// TIA Portal V17 export
// export: Created 2024-06-14T09:52:32.4574024Z, ExportSetting WithDefaults, DisplayName Totally Integrated Automation Portal, DisplayVersion V17, DisplayName TIA Portal Openness, DisplayVersion V17, DisplayName TIA Portal Version Control Interface, DisplayVersion V17, DisplayName Simotion SCOUT TIA, DisplayVersion 5.4.3.0, DisplayName SINAMICS Startdrive Advanced, DisplayVersion V17 SP1 Update 1, DisplayName SINAMICS Startdrive G110M, G120, G120C, G120D, G120P, G115D, DisplayVersion V17 SP1 Update 1, DisplayName SINAMICS Startdrive G130, G150, S120, S150, SINAMICS MV, S210, DisplayVersion V17 SP1 Update 1, DisplayName STEP 7 Professional, DisplayVersion V17, DisplayName STEP 7 Safety, DisplayVersion V17, DisplayName WinCC Professional, DisplayVersion V17
FUNCTION "MODTCP_STN5_FC_L2" : Void   // FC101, LAD
{ S7_Optimized_Access := 'TRUE' }
VERSION : 0.1
// stored: AutoNumber false, IsIECCheckEnabled false, SetENOAutomatically false, UDAEnableTagReadback false
BEGIN

REGION Network 2: Call Filling Line-1 Station-1
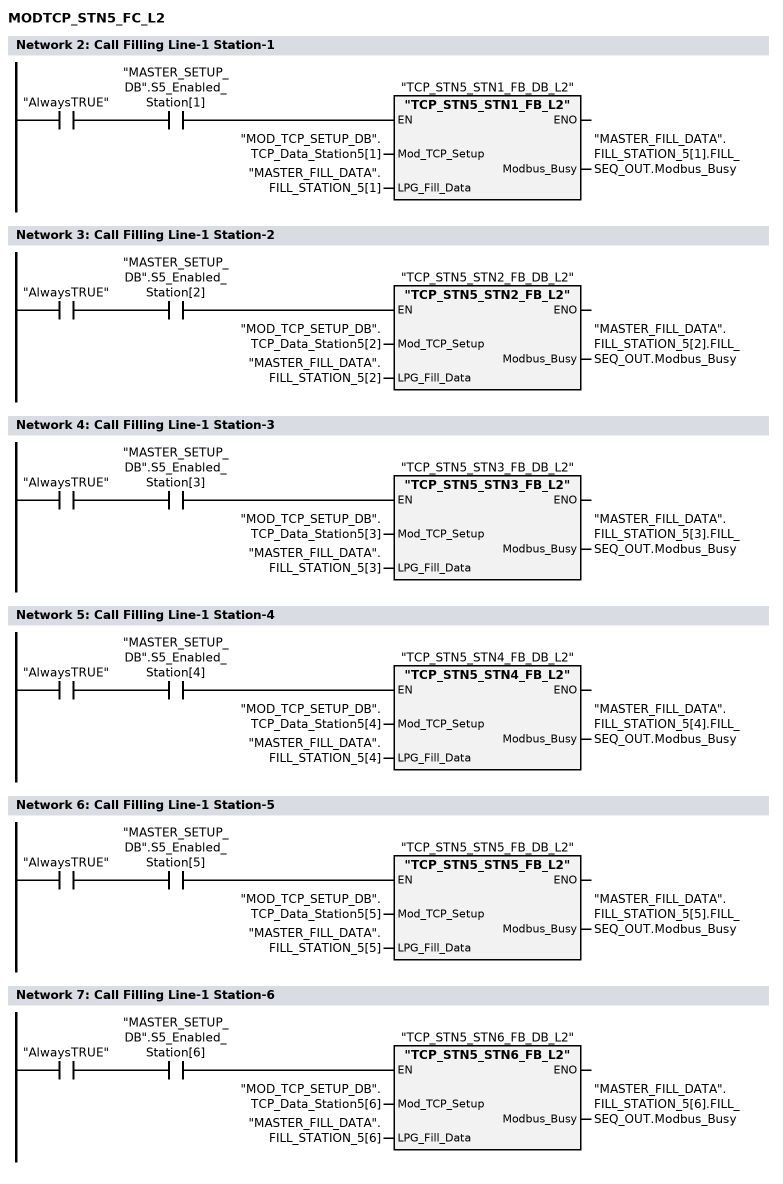
   RUNG wire#powerrail
      Contact( "AlwaysTRUE" )
      Contact( "MASTER_SETUP_DB".S5_Enabled_Station[1] )
      "TCP_STN5_STN1_FB_DB_L2"(Mod_TCP_Setup := "MOD_TCP_SETUP_DB".TCP_Data_Station5[1], LPG_Fill_Data := "MASTER_FILL_DATA".FILL_STATION_5[1], Modbus_Busy => "MASTER_FILL_DATA".FILL_STATION_5[1].FILL_SEQ_OUT.Modbus_Busy)
   END_RUNG
   // the same network as SCL:
   IF "AlwaysTRUE" AND "MASTER_SETUP_DB".S5_Enabled_Station[1] THEN
       "TCP_STN5_STN1_FB_DB_L2"(Mod_TCP_Setup := "MOD_TCP_SETUP_DB".TCP_Data_Station5[1],   // "TCP_STN5_STN1_FB_L2"
                               LPG_Fill_Data := "MASTER_FILL_DATA".FILL_STATION_5[1],
                               Modbus_Busy => "MASTER_FILL_DATA".FILL_STATION_5[1].FILL_SEQ_OUT.Modbus_Busy);
   END_IF;
END_REGION

REGION Network 3: Call Filling Line-1 Station-2
   RUNG wire#powerrail
      Contact( "AlwaysTRUE" )
      Contact( "MASTER_SETUP_DB".S5_Enabled_Station[2] )
      "TCP_STN5_STN2_FB_DB_L2"(Mod_TCP_Setup := "MOD_TCP_SETUP_DB".TCP_Data_Station5[2], LPG_Fill_Data := "MASTER_FILL_DATA".FILL_STATION_5[2], Modbus_Busy => "MASTER_FILL_DATA".FILL_STATION_5[2].FILL_SEQ_OUT.Modbus_Busy)
   END_RUNG
   // the same network as SCL:
   IF "AlwaysTRUE" AND "MASTER_SETUP_DB".S5_Enabled_Station[2] THEN
       "TCP_STN5_STN2_FB_DB_L2"(Mod_TCP_Setup := "MOD_TCP_SETUP_DB".TCP_Data_Station5[2],   // "TCP_STN5_STN2_FB_L2"
                               LPG_Fill_Data := "MASTER_FILL_DATA".FILL_STATION_5[2],
                               Modbus_Busy => "MASTER_FILL_DATA".FILL_STATION_5[2].FILL_SEQ_OUT.Modbus_Busy);
   END_IF;
END_REGION

REGION Network 4: Call Filling Line-1 Station-3
   RUNG wire#powerrail
      Contact( "AlwaysTRUE" )
      Contact( "MASTER_SETUP_DB".S5_Enabled_Station[3] )
      "TCP_STN5_STN3_FB_DB_L2"(Mod_TCP_Setup := "MOD_TCP_SETUP_DB".TCP_Data_Station5[3], LPG_Fill_Data := "MASTER_FILL_DATA".FILL_STATION_5[3], Modbus_Busy => "MASTER_FILL_DATA".FILL_STATION_5[3].FILL_SEQ_OUT.Modbus_Busy)
   END_RUNG
   // the same network as SCL:
   IF "AlwaysTRUE" AND "MASTER_SETUP_DB".S5_Enabled_Station[3] THEN
       "TCP_STN5_STN3_FB_DB_L2"(Mod_TCP_Setup := "MOD_TCP_SETUP_DB".TCP_Data_Station5[3],   // "TCP_STN5_STN3_FB_L2"
                               LPG_Fill_Data := "MASTER_FILL_DATA".FILL_STATION_5[3],
                               Modbus_Busy => "MASTER_FILL_DATA".FILL_STATION_5[3].FILL_SEQ_OUT.Modbus_Busy);
   END_IF;
END_REGION

REGION Network 5: Call Filling Line-1 Station-4
   RUNG wire#powerrail
      Contact( "AlwaysTRUE" )
      Contact( "MASTER_SETUP_DB".S5_Enabled_Station[4] )
      "TCP_STN5_STN4_FB_DB_L2"(Mod_TCP_Setup := "MOD_TCP_SETUP_DB".TCP_Data_Station5[4], LPG_Fill_Data := "MASTER_FILL_DATA".FILL_STATION_5[4], Modbus_Busy => "MASTER_FILL_DATA".FILL_STATION_5[4].FILL_SEQ_OUT.Modbus_Busy)
   END_RUNG
   // the same network as SCL:
   IF "AlwaysTRUE" AND "MASTER_SETUP_DB".S5_Enabled_Station[4] THEN
       "TCP_STN5_STN4_FB_DB_L2"(Mod_TCP_Setup := "MOD_TCP_SETUP_DB".TCP_Data_Station5[4],   // "TCP_STN5_STN4_FB_L2"
                               LPG_Fill_Data := "MASTER_FILL_DATA".FILL_STATION_5[4],
                               Modbus_Busy => "MASTER_FILL_DATA".FILL_STATION_5[4].FILL_SEQ_OUT.Modbus_Busy);
   END_IF;
END_REGION

REGION Network 6: Call Filling Line-1 Station-5
   RUNG wire#powerrail
      Contact( "AlwaysTRUE" )
      Contact( "MASTER_SETUP_DB".S5_Enabled_Station[5] )
      "TCP_STN5_STN5_FB_DB_L2"(Mod_TCP_Setup := "MOD_TCP_SETUP_DB".TCP_Data_Station5[5], LPG_Fill_Data := "MASTER_FILL_DATA".FILL_STATION_5[5], Modbus_Busy => "MASTER_FILL_DATA".FILL_STATION_5[5].FILL_SEQ_OUT.Modbus_Busy)
   END_RUNG
   // the same network as SCL:
   IF "AlwaysTRUE" AND "MASTER_SETUP_DB".S5_Enabled_Station[5] THEN
       "TCP_STN5_STN5_FB_DB_L2"(Mod_TCP_Setup := "MOD_TCP_SETUP_DB".TCP_Data_Station5[5],   // "TCP_STN5_STN5_FB_L2"
                               LPG_Fill_Data := "MASTER_FILL_DATA".FILL_STATION_5[5],
                               Modbus_Busy => "MASTER_FILL_DATA".FILL_STATION_5[5].FILL_SEQ_OUT.Modbus_Busy);
   END_IF;
END_REGION

REGION Network 7: Call Filling Line-1 Station-6
   RUNG wire#powerrail
      Contact( "AlwaysTRUE" )
      Contact( "MASTER_SETUP_DB".S5_Enabled_Station[6] )
      "TCP_STN5_STN6_FB_DB_L2"(Mod_TCP_Setup := "MOD_TCP_SETUP_DB".TCP_Data_Station5[6], LPG_Fill_Data := "MASTER_FILL_DATA".FILL_STATION_5[6], Modbus_Busy => "MASTER_FILL_DATA".FILL_STATION_5[6].FILL_SEQ_OUT.Modbus_Busy)
   END_RUNG
   // the same network as SCL:
   IF "AlwaysTRUE" AND "MASTER_SETUP_DB".S5_Enabled_Station[6] THEN
       "TCP_STN5_STN6_FB_DB_L2"(Mod_TCP_Setup := "MOD_TCP_SETUP_DB".TCP_Data_Station5[6],   // "TCP_STN5_STN6_FB_L2"
                               LPG_Fill_Data := "MASTER_FILL_DATA".FILL_STATION_5[6],
                               Modbus_Busy => "MASTER_FILL_DATA".FILL_STATION_5[6].FILL_SEQ_OUT.Modbus_Busy);
   END_IF;
END_REGION
END_FUNCTION
